Universal Robots PolyScope program: wrs2020_taskboard_belt.urp

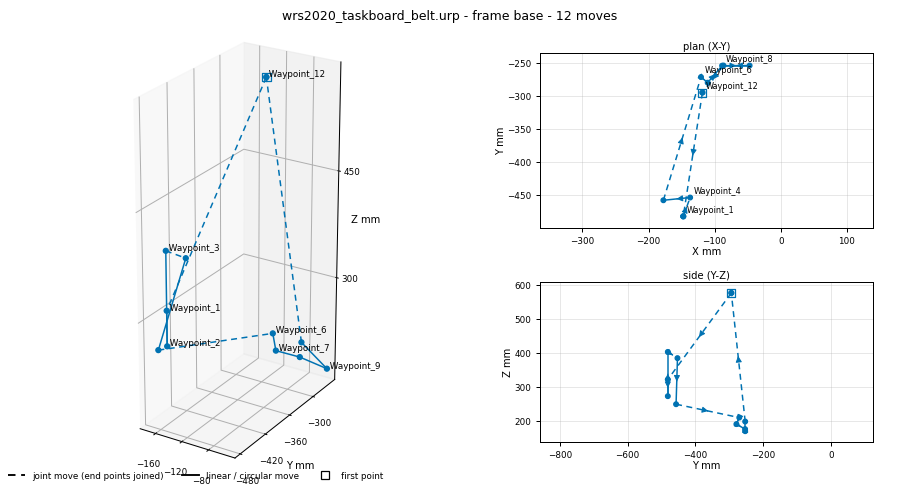
[picture p0: tool path of wrs2020_taskboard_belt.urp in frame base, 12 of 12 moves have a stored position in this frame; points joined in program order, loops and branches not executed]
Program wrs2020_taskboard_belt (installation=default directory=/programs createdIn=5.6.0.90886 lastSavedIn=5.6.0.90886 robotSerialNumber=20205500180)
Calibrated DH parameters: a=[0.000135, -0.030981, -0.334292, 0.000083, 0.000088, 0]; d=[0.162656, 258.79096, -331.603246, 72.945842, 0.099724, 0.099562]; alpha=[1.569535, 0.001639, 0.002824, 1.569633, -1.569323, 0]; deltaTheta=[0, 1.497881, -2.049261, 0.551379, 0, 0]
Robot Program (runOnlyOnce=true)
  MoveJ speed 60 deg/s, acceleration 80 deg/s^2 (useActiveTCP=true) feature=Base
    Waypoint Waypoint_12: TCP in base x=-118.553 y=-294.346 z=577.587 mm, rx=1.3176 ry=2.7241 rz=-0.2718 rad; joints [40.024, -118.444, 99.589, -78.038, -80.282, 2.128] deg
  URCap Gripper (Robotiq_Grippers, Robotiq Inc.) dataModel(position=0.0, force=0.0, speed=0.0, positionInDouble=0.0, forceInDouble=0.0, speedInDouble=0.0, slaveIds=[9], blocking=true)
  MoveJ speed 60 deg/s, acceleration 80 deg/s^2 (useActiveTCP=true) feature=Base
    Waypoint Waypoint_1: TCP in base x=-147.509 y=-481.576 z=322.425 mm, rx=-2.1782 ry=-2.2299 rz=-0.0127 rad; joints [57.916, -85.82, 110.34, -113.684, -91.081, 56.626] deg
    MoveL speed 50 mm/s, acceleration 1200 mm/s^2 (useActiveTCP=true) feature=Base
      Waypoint Waypoint_2: TCP in base x=-147.509 y=-481.576 z=273.212 mm, rx=-2.1897 ry=-2.2414 rz=0.0133 rad; joints [57.763, -82.536, 115.155, -122.915, -90.37, 56.501] deg
  URCap Gripper (Robotiq_Grippers, Robotiq Inc.) dataModel(position=100.0, force=100.0, speed=100.0, positionInDouble=100.0, forceInDouble=100.0, speedInDouble=100.0, slaveIds=[9], blocking=true)
  MoveL speed 250 mm/s, acceleration 1200 mm/s^2 (useActiveTCP=true) feature=Base
    Waypoint Waypoint_3: motionParameters(jointSpeed=1.047198 jointAcceleration=1.396263 cartesianSpeed=0.05 cartesianAcceleration=1.2); TCP in base x=-147.509 y=-481.576 z=403.735 mm, rx=-2.1897 ry=-2.2414 rz=0.0133 rad; joints [57.78, -89.668, 102.124, -102.752, -90.379, 56.451] deg
    MoveJ speed 60 deg/s, acceleration 80 deg/s^2 (useActiveTCP=true) feature=Base
      Waypoint Waypoint_4: TCP in base x=-137.13 y=-453.121 z=385.408 mm, rx=1.7557 ry=1.7734 rz=0.6437 rad; joints [49.802, -89.498, 101.378, -72.762, -56.407, 40.205] deg
  Popup Message (haltProgram=false message=wait for b_bot to move hook into belt inputType=Text)
  MoveL speed 250 mm/s, acceleration 1200 mm/s^2 (useActiveTCP=true) feature=Base
    Waypoint Waypoint_5: TCP in base x=-177.598 y=-457.239 z=249.512 mm, rx=1.4002 ry=1.3073 rz=1.1249 rad; joints [44.345, -69.592, 99.535, -45.535, -45.348, 13.605] deg
  MoveJ speed 60 deg/s, acceleration 80 deg/s^2 (useActiveTCP=true) feature=Base
    Waypoint Waypoint_6: TCP in base x=-120.709 y=-270.878 z=210.116 mm, rx=1.4401 ry=0.8917 rz=0.781 rad; joints [21.225, -92.456, 136.196, -49.18, -40.085, 1.775] deg
  MoveL speed 250 mm/s, acceleration 1200 mm/s^2 (useActiveTCP=true) feature=Base
    Waypoint Waypoint_7: TCP in base x=-110.632 y=-279.411 z=190.846 mm, rx=1.4423 ry=0.8951 rz=0.7781 rad; joints [23.674, -89.974, 137.774, -53.896, -37.643, 2.325] deg
  Popup Message (haltProgram=false message=wait for b_bot to tension inputType=Text)
  MoveL speed 250 mm/s, acceleration 1200 mm/s^2 (useActiveTCP=true) feature=Base
    Waypoint Waypoint_8: TCP in base x=-88.786 y=-253.722 z=176.103 mm, rx=1.479 ry=0.7928 rz=0.6735 rad; joints [18.084, -95.017, 145.843, -56.833, -35.547, 1.971] deg
  MoveL speed 250 mm/s, acceleration 1200 mm/s^2 (useActiveTCP=true) feature=Base
    Waypoint Waypoint_9: TCP in base x=-47.186 y=-253.478 z=169.975 mm, rx=1.5272 ry=0.6376 rz=0.5215 rad; joints [19.093, -103.396, 153.567, -58.237, -23.27, 4.236] deg
  Popup Message (haltProgram=false message=wait for b_bot to thread belt inputType=Text)
  URCap Gripper (Robotiq_Grippers, Robotiq Inc.) dataModel(position=80.3921568627451, force=0.0, speed=0.0, positionInDouble=80.3921568627451, forceInDouble=0.0, speedInDouble=0.0, slaveIds=[9], blocking=true)
  MoveL speed 250 mm/s, acceleration 1200 mm/s^2 (useActiveTCP=true) feature=Base
    Waypoint Waypoint_10: TCP in base x=-86.692 y=-253.478 z=198.507 mm, rx=1.5272 ry=0.6376 rz=0.5215 rad; joints [15.395, -103.398, 147.395, -51.019, -26.952, 3.076] deg
  MoveJ speed 60 deg/s, acceleration 80 deg/s^2 (useActiveTCP=true) feature=Base
    Waypoint Waypoint_11: TCP in base x=-118.553 y=-294.346 z=577.587 mm, rx=1.3176 ry=2.7241 rz=-0.2718 rad; joints [40.024, -118.444, 99.589, -78.038, -80.282, 2.128] deg
